PROGRAM Motormesswerte
VAR
bStart: BOOL := FALSE;	
zaehler : UINT := 0;

//ENC Daten Differenzieren für Geschwindigkeit
diffConst:LREAL:=0.0004;//SECONDS
encDataOldMotor1:UINT:=0;
encDataOldMotor2:UINT:=0;
encDataOldMotor3:UINT:=0;

//Koordinatentransformation Weg
skalEnc:LREAL:=0.00766990393;
x1:LREAL:=0;
x2:LREAL:=0;
x3:LREAL:=0;

xFromMotor1:LREAL:=0;
xFromMotor2:LREAL:=0;
xFromMotor3:LREAL:=0;

//Koordinatentransformation Geschwindigkeit
v1:LREAL:=0;
v2:LREAL:=0;
v3:LREAL:=0;
velocityFromMotor1:LREAL:=0;
velocityFromMotor2:LREAL:=0;
velocityFromMotor3:LREAL:=0;

//INPUTS
encDataFromMotor1 AT%I*  :UINT:=0;
encDataFromMotor2 AT%I*  :UINT:=0;
encDataFromMotor3 AT%I*  :UINT:=0;

diff:  INT :=0;
diff1: INT := 0;
diff2: INT := 0;
diff3: INT := 0;

//OUTPUTS
posXCartesianFromMotors AT%Q*:LREAL:=0;
posYCartesianFromMotors AT%Q*:LREAL:=0;
posThetaCartesianFromMotors AT%Q*:LREAL:=0;

vXCartesianFromMotors AT%Q*:LREAL:=0;
vYCartesianFromMotors AT%Q*:LREAL:=0;
vthetaCartesianFromMotors AT%Q*:LREAL:=0;
END_VAR

IF bStart = FALSE THEN
	encDataOldMotor1 := encDataFromMotor1;
	encDataOldMotor2 := encDataFromMotor2;
	encDataOldMotor3 := encDataFromMotor3;
	bStart := TRUE;
END_IF



// Encoder Wegberechnung und Differenzierung für Geschwindigkeit
diff1:=UINT_TO_INT(encDataFromMotor1) - UINT_TO_INT(encDataOldMotor1);
IF diff1 >= 32767 OR diff1 <= -32767 THEN
	diff1 := 0;
	zaehler := zaehler + 1;
END_IF
diff2:=UINT_TO_INT(encDataFromMotor2) - UINT_TO_INT(encDataOldMotor2);
IF diff2 >= 32767 OR diff2 <= -32767 THEN
	diff2 := 0;
END_IF
diff3:=UINT_TO_INT(encDataFromMotor3) - UINT_TO_INT(encDataOldMotor3);
IF diff3 >= 32767 OR diff3 <= -32767 THEN
	diff3 := 0;
END_IF

xFromMotor1:=xFromMotor1+diff1*skalEnc;
velocityFromMotor1:=diff1/diffConst*skalEnc;

xFromMotor2:=xFromMotor2+diff2*skalEnc;
velocityFromMotor2:=diff2/diffConst*skalEnc;

xFromMotor3:=xFromMotor3+diff3*skalEnc;
velocityFromMotor3:=diff3/diffConst*skalEnc;

// Koordinatentransformation Weg
x1:=-xFromMotor1;
x2:=-xFromMotor2;
x3:=-xFromMotor3;

posXCartesianFromMotors:=(x3 - x1) / (2.0 * COS(30.0*PI/180));  //in mm / s
posYCartesianFromMotors:=(x1 - 2.0 * x2 + x3) / 3.0;            //in mm / s
posThetaCartesianFromMotors:=(x1 + x2 + x3) / (3.0 * 135.0);    //in rad / s

// Koordinatentransformation Geschwindigkeit
v1:=-velocityFromMotor1;
v2:=-velocityFromMotor2;
v3:=-velocityFromMotor3;

vXCartesianFromMotors:=(v3 - v1) / (2.0 * COS(30.0*PI/180));  //in mm / s
vYCartesianFromMotors:=(v1 - 2.0 * v2 + v3) / 3.0;            //in mm / s
vThetaCartesianFromMotors:=(v1 + v2 + v3) / (3.0 * 135.0);    //in rad / s

// Alte Encoderdaten speichern

encDataOldMotor1:=encDataFromMotor1;
encDataOldMotor2:=encDataFromMotor2;
encDataOldMotor3:=encDataFromMotor3;

END_PROGRAM

(* stored: Version 1.1.0.1, ProductVersion 3.1.4022.3
   POU Motormesswerte: Id {bfdecdb6-85cd-45e5-8fd3-068aaa1edc04}, SpecialFunc None *)
